{attribute 'pack_mode' :=  '1'}
TYPE ST_PyADS :
STRUCT
	iInt 	: UINT;
	fReal 	: LREAL;
	aArray  : ARRAY[0..10] OF INT;
END_STRUCT
END_TYPE

(* stored: Version 1.1.0.1, ProductVersion 3.1.4024.12
   DUT ST_PyADS: Id {77746f7b-7901-47c5-8038-69f423560f08} *)
